// TIA Portal project "S7-SCL-P1-E2 Linia sortujaca z waga 5" (V15.1)
// Vorlageprojekt für das Buch mit Zielsystem S7-1200

(* hardware
DEVICE "S71500/ET200MP-Station_1"  S7-1500 station
   slot 0: "Profilschiene_0"  Rack  6ES7 590-1***0-0AA0
   slot 1: "PLC_3"  CPU 1511-1 PN  6ES7 511-1AK00-0AB0  V1.8
      slot 3: "CPU-Display_1"  6ES7591-1AA00-0AA0
   slot 2: "AI 8xU/I/RTD/TC ST_1"  AI 8xU/I/RTD/TC ST  6ES7 531-7KF00-0AB0  V2.0
   slot 3: "AI 8xU/I/RTD/TC ST_2"  AI 8xU/I/RTD/TC ST  6ES7 531-7KF00-0AB0  V2.0
   slot 4: "AI 8xU/I/RTD/TC ST_3"  AI 8xU/I/RTD/TC ST  6ES7 531-7KF00-0AB0  V2.0
   slot 5: "AI 8xU/I/RTD/TC ST_4"  AI 8xU/I/RTD/TC ST  6ES7 531-7KF00-0AB0  V2.0
   slot 6: "DI 16x24VDC BA_1"  DI 16x24VDC BA  6ES7 521-1BH10-0AA0  V1.0
*)

// ===== PLC "PLC_3"  CPU 1511-1 PN =====

VAR_GLOBAL   // PLC tag table "Standard-Variablentabelle"
   "iLicznikTest" AT %MW0 : Int;
END_VAR

VAR_GLOBAL CONSTANT   // PLC tag table "Standard-Variablentabelle"
   "iNA_WPROST" : Int := 0;
   "iPRAWO" : Int := 1;
   "iLEWO" : Int := 2;
END_VAR

VAR_GLOBAL   // PLC tag table "Tag table_1"
   "xSensorWagaWejscie" AT %I0.0 : Bool;
   "xSensorWagaNaSrodku" AT %I0.1 : Bool;
   "xSensorWagaWyjscie" AT %I0.2 : Bool;
   "xStartLight" AT %Q1.0 : Bool;
   "xResetLight" AT %Q1.1 : Bool;
   "xStopLight" AT %Q1.2 : Bool;
   "rWaga" AT %ID30 : Real;
   "diLicznikLewo" AT %QD30 : DInt;
   "diLicznikPrawo" AT %QD38 : DInt;
   "xAuto" AT %I1.4 : Bool;
   "xSensorPodLewyWejscie" AT %I0.3 : Bool;
   "xSensorPodLewyWyjscie" AT %I0.4 : Bool;
   "xSensorPodProstoWejscie" AT %I0.5 : Bool;
   "xSensorPodProstoWyjscie" AT %I0.6 : Bool;
   "xSensorPodPrawyWejscie" AT %I0.7 : Bool;
   "xSensorPodPrawyWyjscie" AT %I1.0 : Bool;
   "xStart" AT %I1.1 : Bool;
   "xStop" AT %I1.3 : Bool;
   "xReset" AT %I1.2 : Bool;
   "diLicznikProsto" AT %QD34 : DInt;
   "rWagaWyswietlacz" AT %QD42 : Real;
   "xPodajnikWej" AT %Q0.0 : Bool;
   "xPodajnikWaga" AT %Q0.1 : Bool;
   "xPodSortLewo" AT %Q0.2 : Bool;
   "xPodajnikLewy" AT %Q0.3 : Bool;
   "xPodSortPrawo" AT %Q0.4 : Bool;
   "xPodajnikPrawy" AT %Q0.5 : Bool;
   "xPodajnikProsto" AT %Q0.7 : Bool;
   "xPodSortWlaczNaped" AT %Q0.6 : Bool;
   "xEstop" AT %I1.5 : Bool;
END_VAR

VAR_GLOBAL CONSTANT   // PLC tag table "Tag table_1"
   "Keiner(1)" : Pip := 65535;
   "Automatische Aktualisierung(1)" : Pip := 0;
   "TPA 1(1)" : Pip := 1;
   "TPA 2(1)" : Pip := 2;
   "TPA 3(1)" : Pip := 3;
   "TPA 4(1)" : Pip := 4;
   "TPA OB Servo(1)" : Pip := 32768;
   "Local~MC(1)" : Hw_SubModule := 51;
   "Local~Common(1)" : Hw_SubModule := 50;
   "Local~Device(1)" : Hw_Device := 32;
   "Local~Configuration(1)" : Hw_SubModule := 33;
   "Local~Exec(1)" : Hw_SubModule := 52;
   "Local(1)" : Hw_SubModule := 49;
   "Local~PROFINET-Schnittstelle_1(1)" : Hw_Interface := 64;
   "Local~PROFINET-Schnittstelle_1~Port_1(1)" : Hw_Interface := 65;
   "Local~HSC_1" : Hw_Hsc := 257;
   "Local~HSC_2" : Hw_Hsc := 258;
   "Local~HSC_3" : Hw_Hsc := 259;
   "Local~HSC_4" : Hw_Hsc := 260;
   "Local~HSC_5" : Hw_Hsc := 261;
   "Local~HSC_6" : Hw_Hsc := 262;
   "Local~AI_2_1" : Hw_SubModule := 263;
   "Local~DI_6_DQ_4_1" : Hw_SubModule := 264;
   "Local~Pulse_1" : Hw_Pwm := 265;
   "Local~Pulse_2" : Hw_Pwm := 266;
   "Local~Pulse_3" : Hw_Pwm := 267;
   "Local~Pulse_4" : Hw_Pwm := 268;
   "OB_Main(1)" : OB_PCYCLE := 1;
   "OB_Cyclic interrupt(2)" : OB_Cyclic := 30;
   "OB_Cyclic interrupt(3)" : OB_Cyclic := 31;
END_VAR

DATA_BLOCK "Linia"   // DB1
{ S7_Optimized_Access := 'TRUE' }
VERSION : 0.1
   VAR
      xAlarmAktywny : Bool;
      xStartLinii : Bool;
      xProduktNaWadze : Bool;
      iPodSortKierunek : Int;
      rWagaAktProduktu : Real;   // [kg]
      aPrzedziałyWagowe : Array[0..2] of Real;
      iLiczbaProbekTest : Int := 20;
      xProduktNaPodSortujacym : Bool;
      wAlarmy : Word;
   END_VAR
BEGIN
   aPrzedziałyWagowe[2] := 17.0;   // [kg]
   aPrzedziałyWagowe[1] := 11.0;   // [kg]
   aPrzedziałyWagowe[0] := 9.0;   // [kg]
END_DATA_BLOCK

DATA_BLOCK "SredniaKroczaca_DB"   // DB5
{ S7_Optimized_Access := 'TRUE' }
VERSION : 0.1
// stored: InstanceOfName SredniaKroczaca
"SredniaKroczaca"
BEGIN
END_DATA_BLOCK

// folder: System blocks/Program resources

DATA_BLOCK "IEC_Timer_WatchDogPodSort"   // DB10
{ S7_Optimized_Access := 'TRUE' }
AUTHOR : Simatic
FAMILY : IEC
NAME : IEC_TMR
VERSION : 1.0
// stored: InstanceOfName IEC_TIMER
"IEC_TIMER"
BEGIN
END_DATA_BLOCK

DATA_BLOCK "IEC_Timer_WatchDogWagi"   // DB11
{ S7_Optimized_Access := 'TRUE' }
AUTHOR : Simatic
FAMILY : IEC
NAME : IEC_TMR
VERSION : 1.0
// stored: InstanceOfName IEC_TIMER
"IEC_TIMER"
BEGIN
END_DATA_BLOCK

DATA_BLOCK "IEC_Counter_LewyTrans"   // DB12
{ S7_Optimized_Access := 'TRUE' }
AUTHOR : Simatic
FAMILY : IEC
NAME : CNTR
VERSION : 1.0
// stored: InstanceOfName IEC_COUNTER
"IEC_COUNTER"
BEGIN
END_DATA_BLOCK

DATA_BLOCK "IEC_Counter_PrawyTran"   // DB14
{ S7_Optimized_Access := 'TRUE' }
AUTHOR : Simatic
FAMILY : IEC
NAME : CNTR
VERSION : 1.0
// stored: InstanceOfName IEC_COUNTER
"IEC_COUNTER"
BEGIN
END_DATA_BLOCK

DATA_BLOCK "IEC_Counter_ProstoTrans"   // DB15
{ S7_Optimized_Access := 'TRUE' }
AUTHOR : Simatic
FAMILY : IEC
NAME : CNTR
VERSION : 1.0
// stored: InstanceOfName IEC_COUNTER
"IEC_COUNTER"
BEGIN
END_DATA_BLOCK

DATA_BLOCK "IEC_Timer_ResetLicznikow"   // DB16
{ S7_Optimized_Access := 'TRUE' }
AUTHOR : Simatic
FAMILY : IEC
NAME : IEC_TMR
VERSION : 1.0
// stored: InstanceOfName IEC_TIMER
"IEC_TIMER"
BEGIN
END_DATA_BLOCK

// folder: (top level)

FUNCTION_BLOCK "SredniaKroczaca"   // FB1, SCL
{ S7_Optimized_Access := 'TRUE' }
VERSION : 0.1
   VAR_INPUT
      rSygnalWejsciowy : Real;
      iLiczbaProbek : Int;
      xStart : Bool;
   END_VAR
   VAR_OUTPUT
      rSygnalWyUsredniony : Real;
      xObliczeniaOK : Bool;
   END_VAR
   VAR
      R_TRIG_Start : R_TRIG;
      aTablicaProbek : Array[0..99] of Real;
   END_VAR
   VAR_TEMP
      rSuma : Real;
      iLicznik : Int;
   END_VAR
BEGIN

   REGION SprawdzenieDLugosciOkna
       IF #iLiczbaProbek < 2 OR #iLiczbaProbek > 100 THEN
           #xObliczeniaOK := 0;
           RETURN;
       END_IF;
   END_REGION


   REGION InicjalizacjaTablicyProbek
       #R_TRIG_Start(CLK := #xStart);

       IF #R_TRIG_Start.Q THEN
           FOR #iLicznik := 0 TO 99 DO // Statement section IF
               #aTablicaProbek[#iLicznik] := 0;
           END_FOR;
       END_IF;
   END_REGION


   REGION ObliczeniaSredniej
       IF #xStart THEN
           // odswiezenie bufora
           FOR #iLicznik := (#iLiczbaProbek - 2) TO 0 BY -1 DO
               #aTablicaProbek[#iLicznik + 1] := #aTablicaProbek[#iLicznik];
               ;
           END_FOR;
           #aTablicaProbek[0] := #rSygnalWejsciowy;

           // obliczenie sumy
           #rSuma := 0;
           FOR #iLicznik := 0 TO #iLiczbaProbek - 1 DO
               #rSuma := #rSuma + #aTablicaProbek[#iLicznik];
           END_FOR;

           // obliczenie sredniej
           #rSygnalWyUsredniony := #rSuma / #iLiczbaProbek;

           // sprawdzenie poprawności obliczeń
           IF ENO THEN
               #xObliczeniaOK := true;
           ELSE
               #xObliczeniaOK := false;
               RETURN;
           END_IF;

       ELSE
           #rSygnalWyUsredniony := 0;
       END_IF;
   END_REGION
END_FUNCTION_BLOCK

FUNCTION "MHJ-PLC-Lab-Function-S71500" : Void   // FC9000, SCL
{ S7_Optimized_Access := 'TRUE' }
VERSION : 0.1
   VAR_TEMP
      Value : Byte;
      ForCounter : Int;
   END_VAR
   VAR CONSTANT
      Value_01_DW : DWord := 16#1223_5486;
      Value_02_DW : DWord := 16#A6C9_D1F5;
   END_VAR
BEGIN

   #Value:=PEEK(area := 16#82,
        dbNumber := 0,
        byteOffset := 511);
   #Value := #Value + 1;

   POKE(area := 16#82,
        dbNumber := 0,
        byteOffset := 511,
        value := #Value);

   POKE(area := 16#82,
        dbNumber := 0,
        byteOffset := 1016,
        value := #Value_01_DW);
   POKE(area := 16#82,
        dbNumber := 0,
        byteOffset := 1020,
        value := #Value_02_DW);

   FOR #ForCounter := 0 TO 63 DO
       #Value:=PEEK(area := 16#1,
            dbNumber := 0,
            byteOffset := #ForCounter);
       POKE(area := 16#81,
            dbNumber := 0,
            byteOffset := #ForCounter,
            value := #Value);
   END_FOR;
   #Value := PEEK(area := 16#1,
                  dbNumber := 0,
                  byteOffset := 512);
   POKE(area := 16#82,
        dbNumber := 0,
        byteOffset := 512,
        value := #Value);
END_FUNCTION

ORGANIZATION_BLOCK "Main"   // OB1, LAD, ProgramCycle
TITLE = "Main Program Sweep (Cycle)"
{ S7_Optimized_Access := 'TRUE' }
VERSION : 0.1
   VAR_INPUT
      Initial_Call : Bool;   // Initial call of this OB
      Remanence : Bool;   // =True, if remanent data are available
   END_VAR
BEGIN
END_ORGANIZATION_BLOCK

ORGANIZATION_BLOCK "ProgramCykliczny"   // OB30, SCL, CyclicInterrupt
{ S7_Optimized_Access := 'TRUE' }
VERSION : 0.1
   VAR_INPUT
      Initial_Call : Bool;   // Initial call of this OB
      Event_Count : Int;   // Events discarded
   END_VAR
   VAR_TEMP
      rTemp_1 : Real;
      iLicznik : Int;
      rSuma : Real;
   END_VAR
BEGIN
   REGION TriggeryOrazTimery
       // triggery podajnika wagowego
       "R_TRIG_WjazdNaWage"(CLK := "xSensorWagaWejscie");
       "F_TRIG_WyjazdzWagi"(CLK := "xSensorWagaWyjscie");
       "F_TRIG_WyjazdLewy"(CLK := "xSensorPodLewyWejscie");
       "F_TRIG_WyjazdPrawy"(CLK := "xSensorPodPrawyWejscie");
       "F_TRIG_WyjazdPrzod"(CLK := "xSensorPodProstoWejscie");
       "R_TRIG_PomiarWaga"(CLK := "xSensorWagaNaSrodku");
       "IEC_Timer_WatchDogPodSort".TON(IN := "Linia".xProduktNaPodSortujacym,
                                       PT := T#2s);
       "IEC_Timer_WatchDogWagi".TON(IN := "Linia".xProduktNaWadze,
                                    PT := T#4s);
   END_REGION

   REGION LicznikiPosortowanychPaczek
       // Wyswietlanie licznikow posortowanych paczek i ich resetowanie
       "IEC_Timer_ResetLicznikow".TON(IN:=NOT "xStop",
                                      PT:=T#3s);

       "IEC_Counter_LewyTrans".CTU(CU := "xSensorPodLewyWyjscie",
                                   R := "IEC_Timer_ResetLicznikow".Q,
                                   PV := 1000,
                                   CV => "diLicznikLewo");
       "IEC_Counter_PrawyTran".CTU(CU := "xSensorPodPrawyWyjscie",
                                   R:="IEC_Timer_ResetLicznikow".Q,
                                   PV := 1000,
                                   CV => "diLicznikPrawo");
       "IEC_Counter_ProstoTrans".CTU(CU := "xSensorPodProstoWyjscie",
                                     R:="IEC_Timer_ResetLicznikow".Q,
                                     PV := 1000,
                                     CV => "diLicznikProsto");
   END_REGION

   REGION ObsługaWagi
       "SredniaKroczaca_DB"(rSygnalWejsciowy := "rWaga",
                            iLiczbaProbek := "Linia".iLiczbaProbekTest,
                            xStart := true);

       IF "R_TRIG_PomiarWaga".Q THEN
           // skalowanie z 0-10.0 V na 0-20.0 kg
           "Linia".rWagaAktProduktu := "SredniaKroczaca_DB".rSygnalWyUsredniony * REAL#2.0;
           // wyswietlenie wartości 0-10.0 V sygnału uśrednionego z wagi
           "rWagaWyswietlacz" := "SredniaKroczaca_DB".rSygnalWyUsredniony;
       END_IF;
   END_REGION


   REGION UkladStartStop
       "R_TRIG_Start"(CLK := "xStart");

       IF NOT "xStop" OR NOT "xEstop" OR "Linia".xAlarmAktywny THEN
           "Linia".xStartLinii := FALSE;
       ELSIF "R_TRIG_Start".Q THEN
           "Linia".xStartLinii := true;
       END_IF;

       "xStartLight" := "Linia".xStartLinii;
       "xStopLight" := NOT "Linia".xStartLinii;
       "xResetLight" := "Linia".xAlarmAktywny;
   END_REGION

   REGION KierunekZjazduPaczkiNaPodstawieWagi
       // okreslenie kierunku na podstawie wagi
       IF "Linia".rWagaAktProduktu < "Linia".aPrzedziałyWagowe[0] THEN
           "Linia".iPodSortKierunek := "iLEWO";
       ELSIF "Linia".rWagaAktProduktu < "Linia".aPrzedziałyWagowe[1] THEN
           "Linia".iPodSortKierunek := "iNA_WPROST";
       ELSIF "Linia".rWagaAktProduktu < "Linia".aPrzedziałyWagowe[2] THEN
           "Linia".iPodSortKierunek := "iPRAWO";
       ELSE
           "Linia".iPodSortKierunek := -1;
       END_IF;
   END_REGION

   REGION SterowaniePodajnikami
       IF "Linia".xStartLinii THEN // tryb start linii
           // załączenie podajników
           "xPodajnikLewy" := 1;
           "xPodajnikPrawy" := 1;
           "xPodajnikProsto" := 1;
           "xPodajnikWaga" := 1;

           // podajnik sortujący
           CASE "Linia".iPodSortKierunek OF
               "iNA_WPROST":
                   "xPodSortLewo" := 0;
                   "xPodSortPrawo" := 0;
                   "xPodSortWlaczNaped" := 1;
                   IF "F_TRIG_WyjazdzWagi".Q THEN
                       "Linia".xProduktNaPodSortujacym := 1;
                   ELSIF "F_TRIG_WyjazdPrzod".Q THEN
                       "Linia".xProduktNaPodSortujacym := 0;
                   END_IF;
               "iPRAWO":
                   "xPodSortLewo" := 0;
                   "xPodSortPrawo" := 1;
                   "xPodSortWlaczNaped" := 1;
                   IF "F_TRIG_WyjazdzWagi".Q THEN
                       "Linia".xProduktNaPodSortujacym := 1;
                   ELSIF "F_TRIG_WyjazdPrawy".Q THEN
                       "Linia".xProduktNaPodSortujacym := 0;
                   END_IF;
               "iLEWO":
                   "xPodSortLewo" := 1;
                   "xPodSortPrawo" := 0;
                   "xPodSortWlaczNaped" := 1;
                   IF "F_TRIG_WyjazdzWagi".Q THEN
                       "Linia".xProduktNaPodSortujacym := 1;
                   ELSIF "F_TRIG_WyjazdLewy".Q THEN
                       "Linia".xProduktNaPodSortujacym := 0;
                   END_IF;
               ELSE
                   "xPodSortLewo" := 0;
                   "xPodSortPrawo" := 0;
                   "xPodSortWlaczNaped" := 0;
           END_CASE;

           // przerzutnik obecności produktu na wadze
           IF "R_TRIG_WjazdNaWage".Q AND NOT #Initial_Call THEN
               "Linia".xProduktNaWadze := 1;
           ELSIF "F_TRIG_WyjazdzWagi".Q THEN
               "Linia".xProduktNaWadze := 0;
           END_IF;

           // ząłączenie podajnika wejściowego
           "xPodajnikWej" := NOT "Linia".xProduktNaWadze OR "xSensorWagaWejscie";

       ELSIF NOT "Linia".xStartLinii THEN  // linia wyłączona
           // wyłączenie podajników
           "xPodajnikLewy" := 0;
           "xPodajnikPrawy" := 0;
           "xPodajnikProsto" := 0;
           "xPodSortWlaczNaped" := 0;
           "xPodajnikWaga" := 0;
           "xPodajnikWej" := 0;

           // reset bitów pamięci stanowiska
           "Linia".xProduktNaWadze := 0;
           "Linia".xProduktNaPodSortujacym := 0;
       END_IF;
   END_REGION

   ;
   REGION AlarmyPrzekroczeniaCzasuiZłegoKierunku
       //Trzy alarmy dotyczące przekroczenia czasu lub przekroczenia złego czujnika
       IF "Linia".iPodSortKierunek = "iPRAWO" AND ("IEC_Timer_WatchDogPodSort".Q OR "xSensorPodLewyWejscie" OR "xSensorPodProstoWejscie") THEN
           "Linia".wAlarmy.%X0 := 1;
       ELSIF "xReset" THEN
           "Linia".wAlarmy.%X0 := 0;
       END_IF;
       IF "Linia".iPodSortKierunek = "iLEWO" AND ("IEC_Timer_WatchDogPodSort".Q OR "xSensorPodPrawyWejscie" OR "xSensorPodProstoWejscie") THEN
           "Linia".wAlarmy.%X1 := 1;
       ELSIF "xReset" THEN
           "Linia".wAlarmy.%X1 := 0;
       END_IF;

       IF "Linia".iPodSortKierunek = "iNA_WPROST" AND ("IEC_Timer_WatchDogPodSort".Q OR "xSensorPodLewyWejscie" OR "xSensorPodPrawyWejscie") THEN
           "Linia".wAlarmy.%X2 := 1;
       ELSIF "xReset" THEN
           "Linia".wAlarmy.%X2 := 0;
       END_IF;
   END_REGION

   REGION AlarmNiewłaściwaWagaPaczki
       //alarm o niewłaściwej wadze paczki
       IF "Linia".iPodSortKierunek = -1 THEN
           "Linia".wAlarmy.%X3 := 1;
       ELSIF "xReset" THEN
           "Linia".wAlarmy.%X3 := 0;
       END_IF;
   END_REGION

   REGION AlarmPrzekroczeniCzasuNaWadze
       //alarm zbyt długiego przebywania produktu na wadze
       IF "IEC_Timer_WatchDogWagi".Q THEN
           "Linia".wAlarmy.%X4 := 1;
       ELSIF "xReset" THEN
           "Linia".wAlarmy.%X4 := 0;
       END_IF;
   END_REGION


   REGION AktywacjaAlarmu
       IF "Linia".wAlarmy <> 0 THEN
           "Linia".xAlarmAktywny := 1;
       ELSE
           "Linia".xAlarmAktywny := 0;
       END_IF;
   END_REGION


   "MHJ-PLC-Lab-Function-S71500"();
END_ORGANIZATION_BLOCK